Staubli VAL3: instrSequential.pjx

Parameters version=s7.2.1 stackSize=5000 millimeterUnit=true
Data file=instrSequential.dtx
